(* Logix 5000 project; controller HP_SSC01 vendor 1 type 14 code 67 rev 17.7; software revision 17.01; part 6 of 15 *)
(* tags used below, declared in another part *)
   A_C2_0218 : ALIAS FOR S_C2_FaultSafety.18;
   A_C2_0219 : ALIAS FOR S_C2_FaultSafety.19;
   A_C2_0220 : ALIAS FOR S_C2_FaultSafety.20;
   A_C2_0221 : ALIAS FOR S_C2_FaultSafety.21;
   A_C2_0222 : ALIAS FOR S_C2_FaultSafety.22;
   A_C2_0223 : ALIAS FOR S_C2_FaultSafety.23;
   A_C2_0311 : ALIAS FOR C2_FaultStandard.11;
   A_C2_0312 : ALIAS FOR C2_FaultStandard.12;
   A_C2_0313 : ALIAS FOR C2_FaultStandard.13;
   A_C2_0314 : ALIAS FOR C2_FaultStandard.14;
   A_C2_0315 : ALIAS FOR C2_FaultStandard.15;
   C2 : AXIS_SERVO_DRIVE;
   C2_EncoderDegree : REAL;
   C2_EncoderPositionAtHome : DINT;
   C2_ExcecutePBHoldTimer : TIMER;
   C2_FaultHomeSwitchNotFound : BOOL;
   C2_Homed : BOOL;
   C2_HomeDelay : TIMER[8];
   C2_HomeFindSwitchMAM01 : MOTION_INSTRUCTION;
   C2_HomeFindSwitchMAM02 : MOTION_INSTRUCTION;
   C2_HomeFindSwitchMAS01 : MOTION_INSTRUCTION;
   C2_HomeGetCloseToSwitchMAM01 : MOTION_INSTRUCTION;
   C2_HomeGoToOnPathMAM01 : MOTION_INSTRUCTION;
   C2_HomeMessageNumber : DINT;
   C2_HomeSensorTestMAM02 : MOTION_INSTRUCTION;
   C2_HomeSequence : DINT;
   C2_HomeSequenceAlarms : DINT;
   C2_HomeSequenceAlarmTimer : TIMER[32];
   C2_HomeSequenceInProcess : BOOL;
   C2_HomeSequenceMAH : MOTION_INSTRUCTION;
   C2_HomeSwitchFaultK7KFailedOff : BOOL;
   C2_HomeSwitchFaultK7KFailedOn : BOOL;
   C2_HomeSwitchFaultSafeFailedOff : BOOL;
   C2_HomeSwitchFaultSafeFailedOn : BOOL;
   C2_HomeTest : REAL;
   C2_IndexEnable : BOOL;
   C2_IndexEnableTOF : TIMER;
   C2_IndexMAM01 : MOTION_INSTRUCTION;
   C2_IndexMAS01 : MOTION_INSTRUCTION;
   C2_IndexMessageNumber : DINT;
   C2_IndexPermissive : BOOL;
   C2_Jog_ONS : DINT;
   C2_JogDirection : DINT;
   C2_JogEnable : BOOL;
   C2_JogEnableTOF : TIMER;
   C2_JogForwardFastSelected : BOOL;
   C2_JogForwardSlowSelected : BOOL;
   C2_JogMAJ01 : MOTION_INSTRUCTION;
   C2_JogMAJ02 : MOTION_INSTRUCTION;
   C2_JogMAS01 : MOTION_INSTRUCTION;
   C2_JogMessageNumber : DINT;
   C2_JogPermissive : BOOL;
   C2_JogReverseFastSelected : BOOL;
   C2_JogReverseSlowSelected : BOOL;
   C2_MAJAcceleration : REAL;
   C2_MAJDeceleration : REAL;
   C2_MAJSpeed : REAL;
   C2_OIT_Current : DINT;
   C2_RemoteHomeCMD : BOOL;
   C2_ServoActionStatusOnDelay : TIMER;
   C2_SetEncoderHomePosition : BOOL;
   C2HomeSensorTestMAM01 : MOTION_INSTRUCTION;
   C2HomeSequenceONS : BOOL;
   C2HomeSequenceONS2 : BOOL;
   S_C2_EncoderPositionAtHomeSet : BOOL;
   S_C2_ExecutePB : BOOL;
   S_C2_FaultReset : BOOL;
   S_C2_HomeSafePE : ALIAS FOR C2_Safe:I.Pt04Data;
   S_C2_ModeLocal : BOOL;
   S_C2_ModeRemote : BOOL;
   S_C2_MSTOP_InputOK : BOOL;
   S_EncoderCtsFor360Deg : DINT;
(* Carousel2, continued *)

ROUTINE C230_Home   (* ladder *)
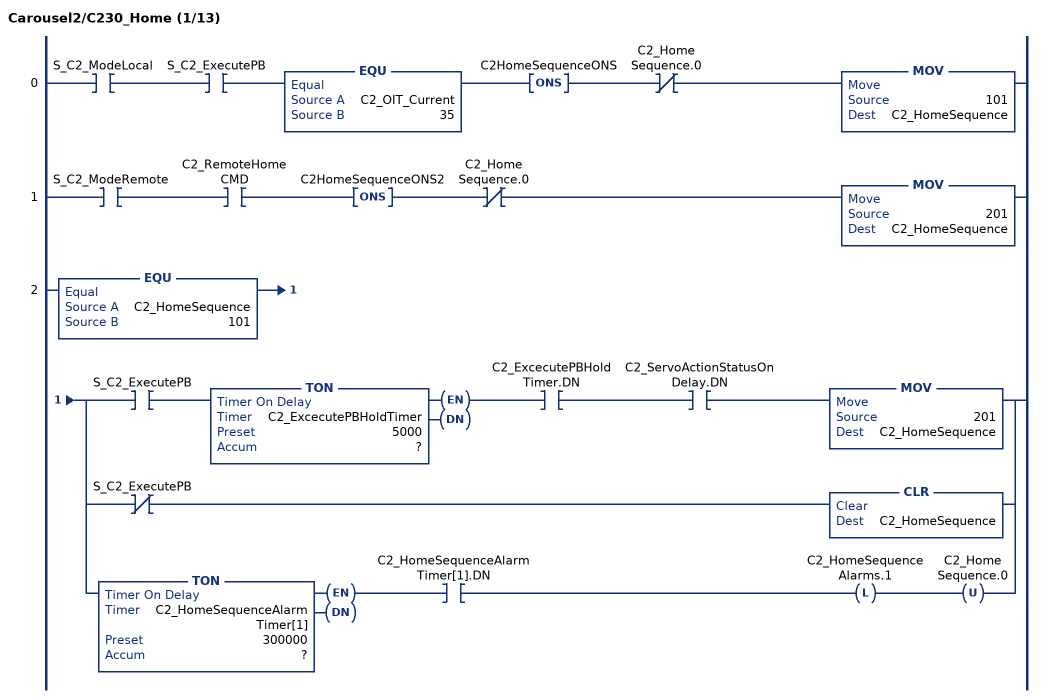
   0: XIC(S_C2_ModeLocal)XIC(S_C2_ExecutePB)EQU(C2_OIT_Current,35)ONS(C2HomeSequenceONS)XIO(C2_HomeSequence.0)MOV(101,C2_HomeSequence);
   1: XIC(S_C2_ModeRemote)XIC(C2_RemoteHomeCMD)ONS(C2HomeSequenceONS2)XIO(C2_HomeSequence.0)MOV(201,C2_HomeSequence);
   2: EQU(C2_HomeSequence,101)[XIC(S_C2_ExecutePB) TON(C2_ExcecutePBHoldTimer,?,?) XIC(C2_ExcecutePBHoldTimer.DN) XIC(C2_ServoActionStatusOnDelay.DN) MOV(201,C2_HomeSequence) ,XIO(S_C2_ExecutePB) CLR(C2_HomeSequence) ,TON(C2_HomeSequenceAlarmTimer[1],?,?) XIC(C2_HomeSequenceAlarmTimer[1].DN) OTL(C2_HomeSequenceAlarms.1) OTU(C2_HomeSequence.0) ];
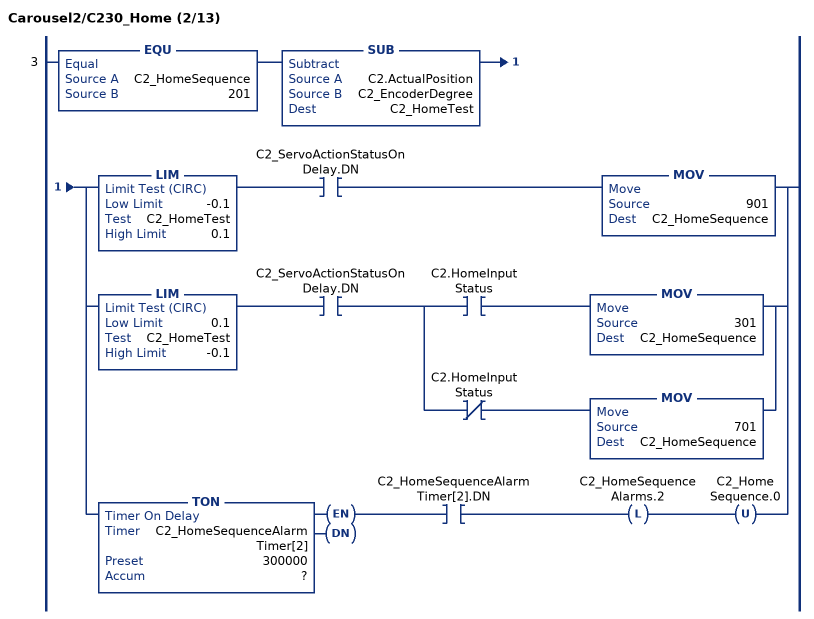
   3: EQU(C2_HomeSequence,201)SUB(C2.ActualPosition,C2_EncoderDegree,C2_HomeTest)[LIM(-0.1,C2_HomeTest,0.1) XIC(C2_ServoActionStatusOnDelay.DN) MOV(901,C2_HomeSequence) ,LIM(0.1,C2_HomeTest,-0.1) XIC(C2_ServoActionStatusOnDelay.DN) [XIC(C2.HomeInputStatus) MOV(301,C2_HomeSequence) ,XIO(C2.HomeInputStatus) MOV(701,C2_HomeSequence) ] ,TON(C2_HomeSequenceAlarmTimer[2],?,?) XIC(C2_HomeSequenceAlarmTimer[2].DN) OTL(C2_HomeSequenceAlarms.2) OTU(C2_HomeSequence.0) ];
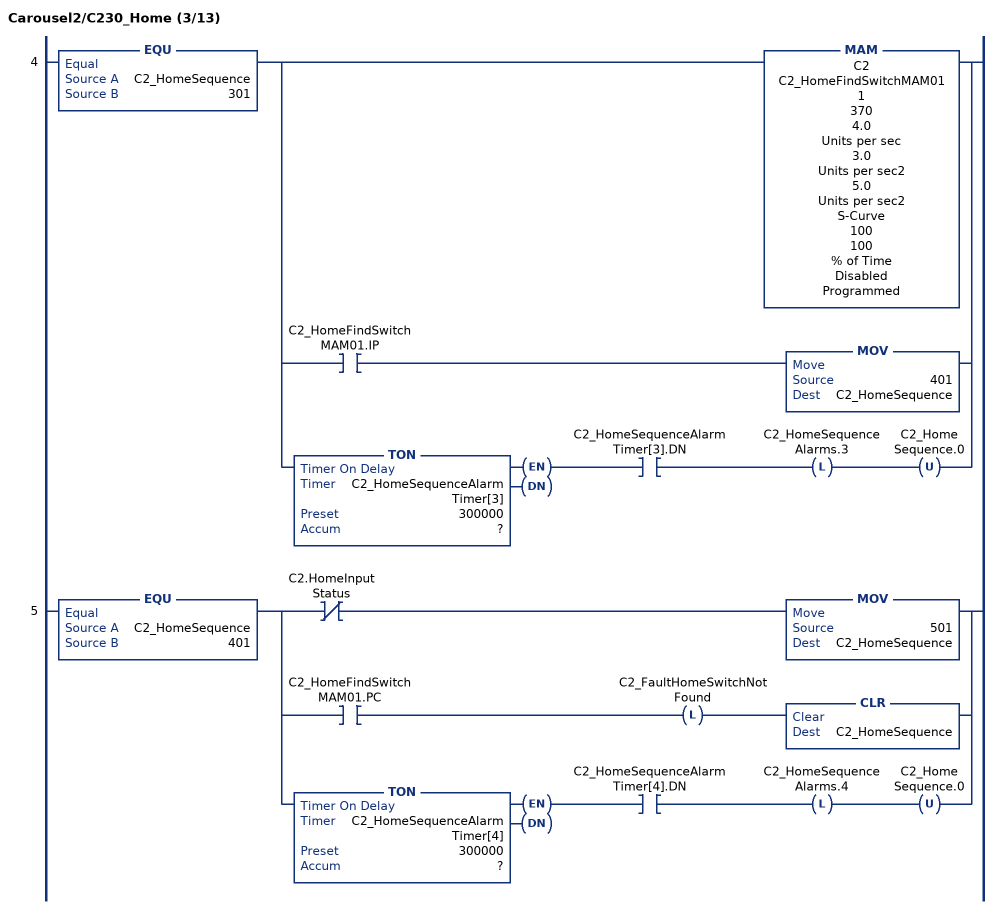
   4: EQU(C2_HomeSequence,301)[MAM(C2,C2_HomeFindSwitchMAM01,1,370,4.0,Units per sec,3.0,Units per sec2,5.0,Units per sec2,S-Curve,100,100,% of Time,Disabled,Programmed) ,XIC(C2_HomeFindSwitchMAM01.IP) MOV(401,C2_HomeSequence) ,TON(C2_HomeSequenceAlarmTimer[3],?,?) XIC(C2_HomeSequenceAlarmTimer[3].DN) OTL(C2_HomeSequenceAlarms.3) OTU(C2_HomeSequence.0) ];
   5: EQU(C2_HomeSequence,401)[XIO(C2.HomeInputStatus) MOV(501,C2_HomeSequence) ,XIC(C2_HomeFindSwitchMAM01.PC) OTL(C2_FaultHomeSwitchNotFound) CLR(C2_HomeSequence) ,TON(C2_HomeSequenceAlarmTimer[4],?,?) XIC(C2_HomeSequenceAlarmTimer[4].DN) OTL(C2_HomeSequenceAlarms.4) OTU(C2_HomeSequence.0) ];
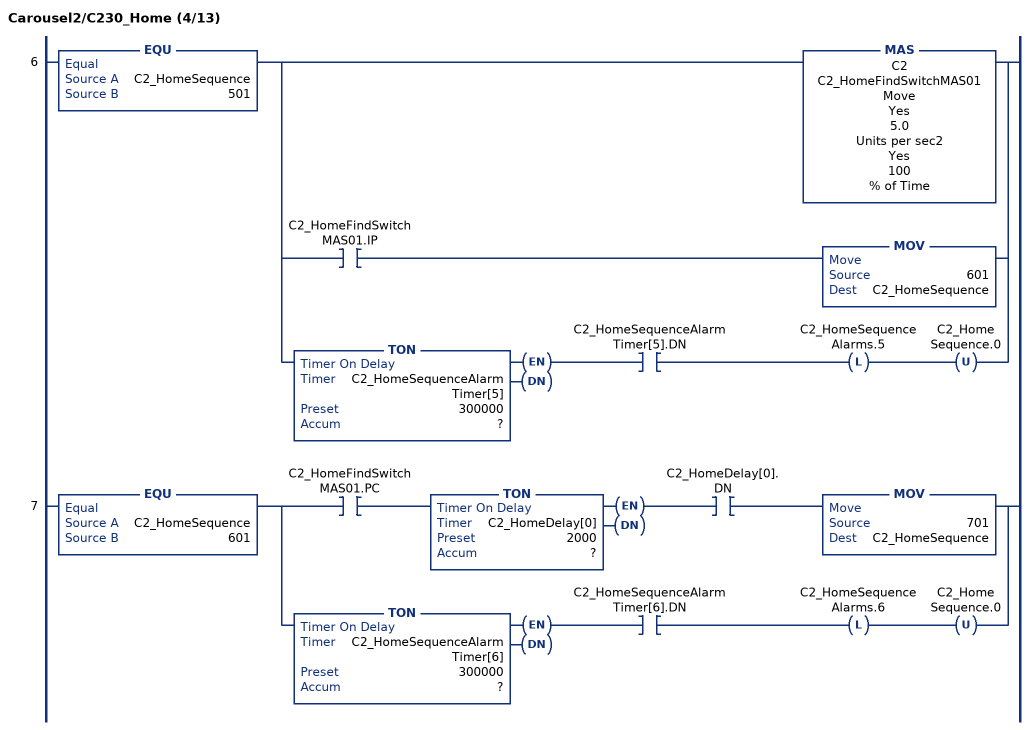
   6: EQU(C2_HomeSequence,501)[MAS(C2,C2_HomeFindSwitchMAS01,Move,Yes,5.0,Units per sec2,Yes,100,% of Time) ,XIC(C2_HomeFindSwitchMAS01.IP) MOV(601,C2_HomeSequence) ,TON(C2_HomeSequenceAlarmTimer[5],?,?) XIC(C2_HomeSequenceAlarmTimer[5].DN) OTL(C2_HomeSequenceAlarms.5) OTU(C2_HomeSequence.0) ];
   7: EQU(C2_HomeSequence,601)[XIC(C2_HomeFindSwitchMAS01.PC) TON(C2_HomeDelay[0],?,?) XIC(C2_HomeDelay[0].DN) MOV(701,C2_HomeSequence) ,TON(C2_HomeSequenceAlarmTimer[6],?,?) XIC(C2_HomeSequenceAlarmTimer[6].DN) OTL(C2_HomeSequenceAlarms.6) OTU(C2_HomeSequence.0) ];
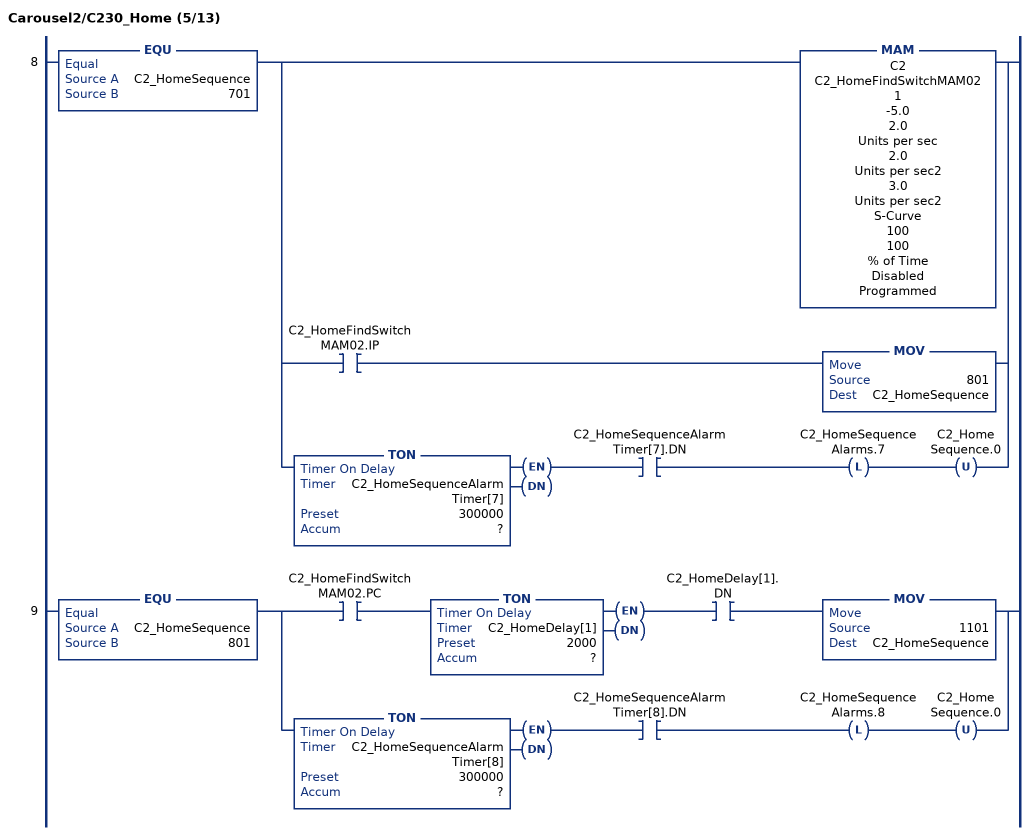
   8: EQU(C2_HomeSequence,701)[MAM(C2,C2_HomeFindSwitchMAM02,1,-5.0,2.0,Units per sec,2.0,Units per sec2,3.0,Units per sec2,S-Curve,100,100,% of Time,Disabled,Programmed) ,XIC(C2_HomeFindSwitchMAM02.IP) MOV(801,C2_HomeSequence) ,TON(C2_HomeSequenceAlarmTimer[7],?,?) XIC(C2_HomeSequenceAlarmTimer[7].DN) OTL(C2_HomeSequenceAlarms.7) OTU(C2_HomeSequence.0) ];
   9: EQU(C2_HomeSequence,801)[XIC(C2_HomeFindSwitchMAM02.PC) TON(C2_HomeDelay[1],?,?) XIC(C2_HomeDelay[1].DN) MOV(1101,C2_HomeSequence) ,TON(C2_HomeSequenceAlarmTimer[8],?,?) XIC(C2_HomeSequenceAlarmTimer[8].DN) OTL(C2_HomeSequenceAlarms.8) OTU(C2_HomeSequence.0) ];
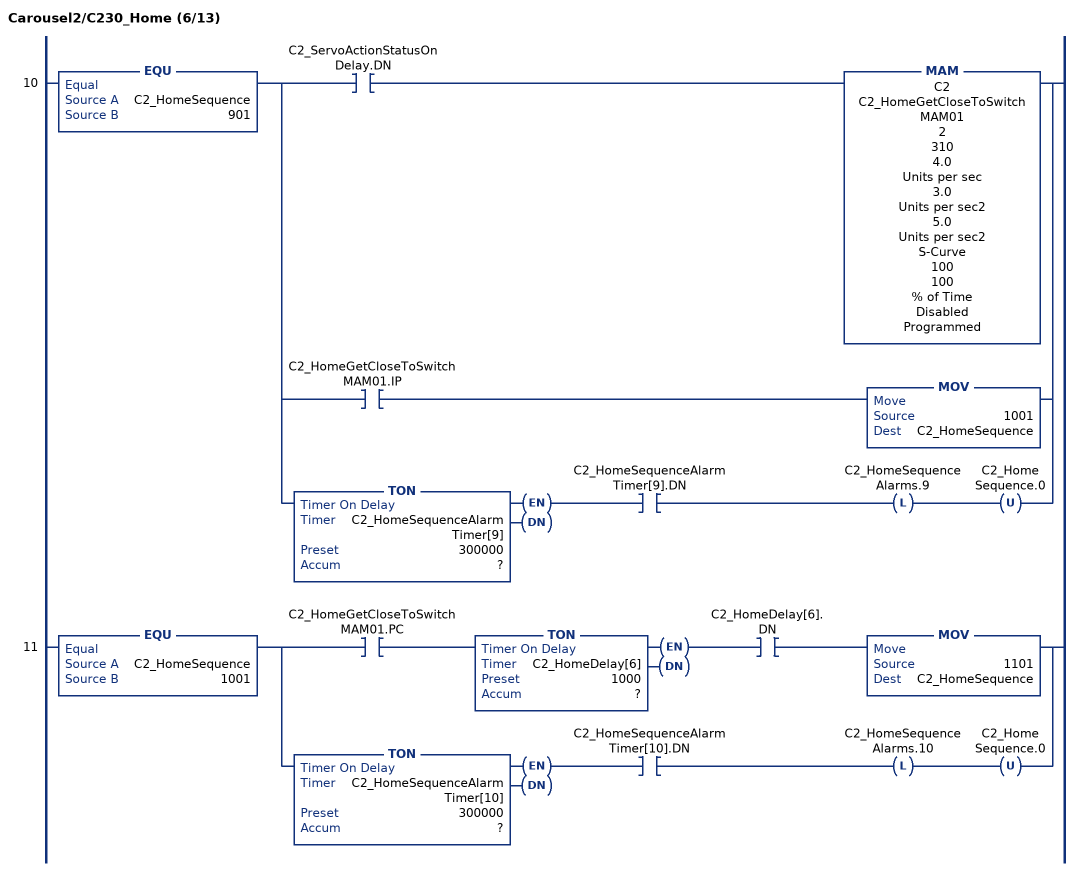
   10: EQU(C2_HomeSequence,901)[XIC(C2_ServoActionStatusOnDelay.DN) MAM(C2,C2_HomeGetCloseToSwitchMAM01,2,310,4.0,Units per sec,3.0,Units per sec2,5.0,Units per sec2,S-Curve,100,100,% of Time,Disabled,Programmed) ,XIC(C2_HomeGetCloseToSwitchMAM01.IP) MOV(1001,C2_HomeSequence) ,TON(C2_HomeSequenceAlarmTimer[9],?,?) XIC(C2_HomeSequenceAlarmTimer[9].DN) OTL(C2_HomeSequenceAlarms.9) OTU(C2_HomeSequence.0) ];
   11: EQU(C2_HomeSequence,1001)[XIC(C2_HomeGetCloseToSwitchMAM01.PC) TON(C2_HomeDelay[6],?,?) XIC(C2_HomeDelay[6].DN) MOV(1101,C2_HomeSequence) ,TON(C2_HomeSequenceAlarmTimer[10],?,?) XIC(C2_HomeSequenceAlarmTimer[10].DN) OTL(C2_HomeSequenceAlarms.10) OTU(C2_HomeSequence.0) ];
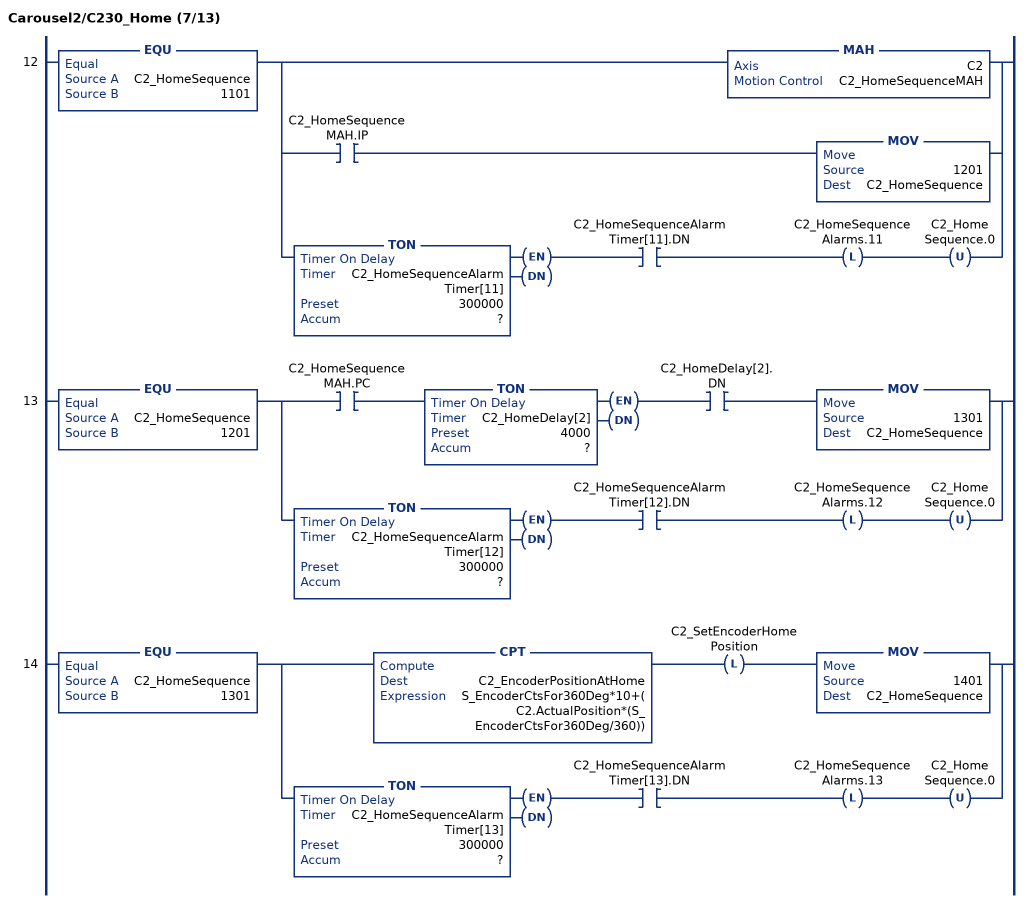
   12: EQU(C2_HomeSequence,1101)[MAH(C2,C2_HomeSequenceMAH) ,XIC(C2_HomeSequenceMAH.IP) MOV(1201,C2_HomeSequence) ,TON(C2_HomeSequenceAlarmTimer[11],?,?) XIC(C2_HomeSequenceAlarmTimer[11].DN) OTL(C2_HomeSequenceAlarms.11) OTU(C2_HomeSequence.0) ];
   13: EQU(C2_HomeSequence,1201)[XIC(C2_HomeSequenceMAH.PC) TON(C2_HomeDelay[2],?,?) XIC(C2_HomeDelay[2].DN) MOV(1301,C2_HomeSequence) ,TON(C2_HomeSequenceAlarmTimer[12],?,?) XIC(C2_HomeSequenceAlarmTimer[12].DN) OTL(C2_HomeSequenceAlarms.12) OTU(C2_HomeSequence.0) ];
   14: EQU(C2_HomeSequence,1301)[CPT(C2_EncoderPositionAtHome,S_EncoderCtsFor360Deg*10+(C2.ActualPosition*(S_EncoderCtsFor360Deg/360))) OTL(C2_SetEncoderHomePosition) MOV(1401,C2_HomeSequence) ,TON(C2_HomeSequenceAlarmTimer[13],?,?) XIC(C2_HomeSequenceAlarmTimer[13].DN) OTL(C2_HomeSequenceAlarms.13) OTU(C2_HomeSequence.0) ];
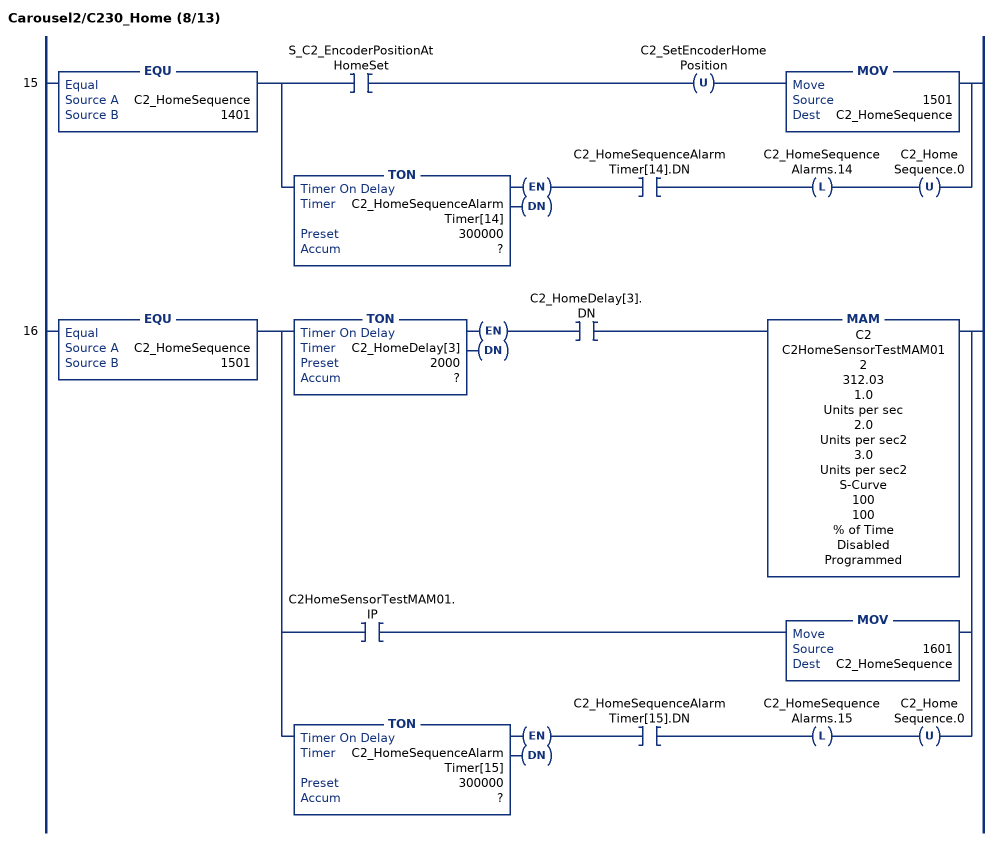
   15: EQU(C2_HomeSequence,1401)[XIC(S_C2_EncoderPositionAtHomeSet) OTU(C2_SetEncoderHomePosition) MOV(1501,C2_HomeSequence) ,TON(C2_HomeSequenceAlarmTimer[14],?,?) XIC(C2_HomeSequenceAlarmTimer[14].DN) OTL(C2_HomeSequenceAlarms.14) OTU(C2_HomeSequence.0) ];
   16: EQU(C2_HomeSequence,1501)[TON(C2_HomeDelay[3],?,?) XIC(C2_HomeDelay[3].DN) MAM(C2,C2HomeSensorTestMAM01,2,312.03,1.0,Units per sec,2.0,Units per sec2,3.0,Units per sec2,S-Curve,100,100,% of Time,Disabled,Programmed) ,XIC(C2HomeSensorTestMAM01.IP) MOV(1601,C2_HomeSequence) ,TON(C2_HomeSequenceAlarmTimer[15],?,?) XIC(C2_HomeSequenceAlarmTimer[15].DN) OTL(C2_HomeSequenceAlarms.15) OTU(C2_HomeSequence.0) ];
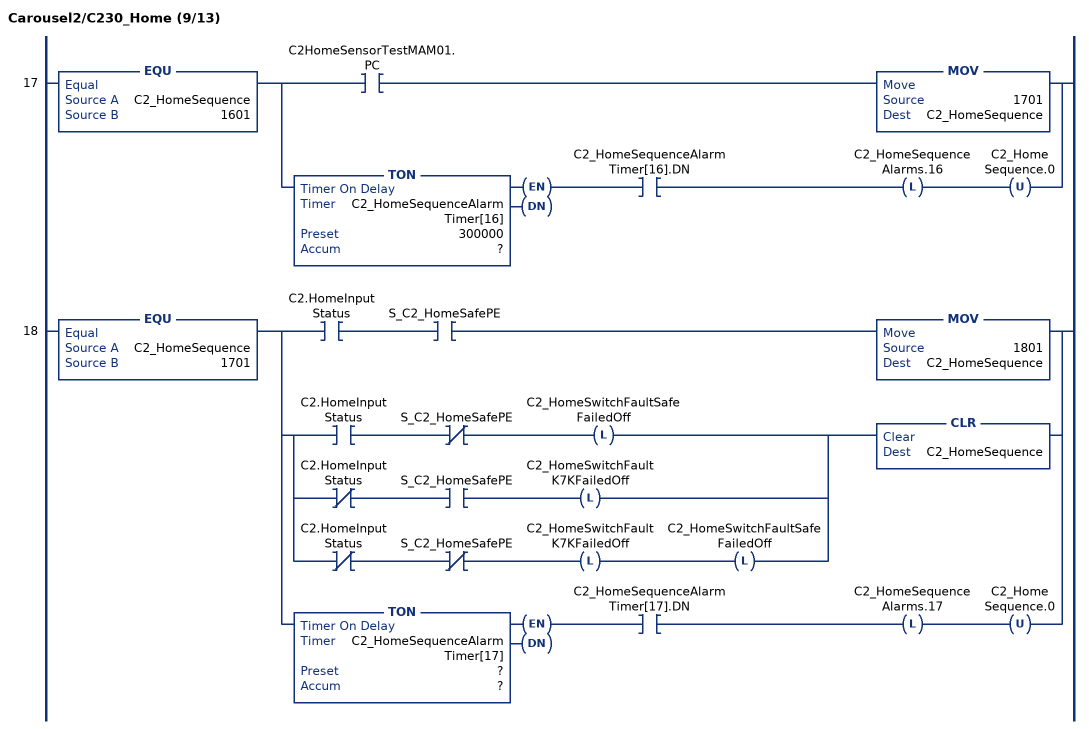
   17: EQU(C2_HomeSequence,1601)[XIC(C2HomeSensorTestMAM01.PC) MOV(1701,C2_HomeSequence) ,TON(C2_HomeSequenceAlarmTimer[16],?,?) XIC(C2_HomeSequenceAlarmTimer[16].DN) OTL(C2_HomeSequenceAlarms.16) OTU(C2_HomeSequence.0) ];
   18: EQU(C2_HomeSequence,1701)[XIC(C2.HomeInputStatus) XIC(S_C2_HomeSafePE) MOV(1801,C2_HomeSequence) ,[XIC(C2.HomeInputStatus) XIO(S_C2_HomeSafePE) OTL(C2_HomeSwitchFaultSafeFailedOff) ,XIO(C2.HomeInputStatus) XIC(S_C2_HomeSafePE) OTL(C2_HomeSwitchFaultK7KFailedOff) ,XIO(C2.HomeInputStatus) XIO(S_C2_HomeSafePE) OTL(C2_HomeSwitchFaultK7KFailedOff) OTL(C2_HomeSwitchFaultSafeFailedOff) ] CLR(C2_HomeSequence) ,TON(C2_HomeSequenceAlarmTimer[17],?,?) XIC(C2_HomeSequenceAlarmTimer[17].DN) OTL(C2_HomeSequenceAlarms.17) OTU(C2_HomeSequence.0) ];
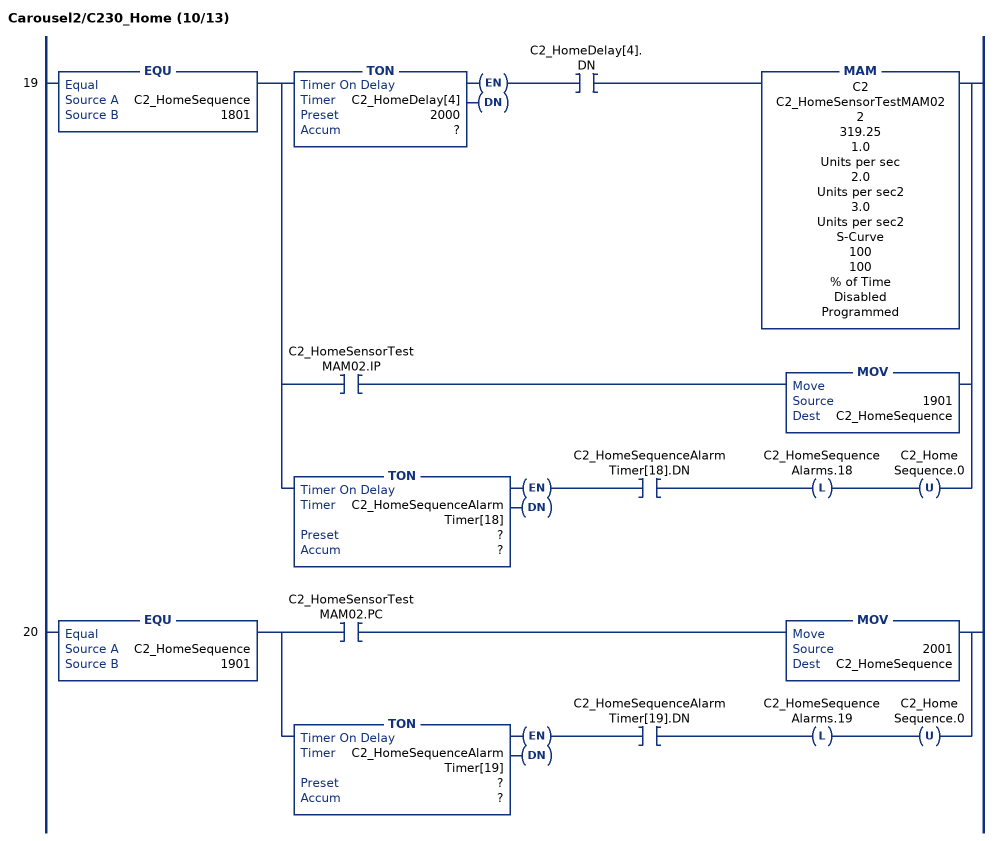
   19: EQU(C2_HomeSequence,1801)[TON(C2_HomeDelay[4],?,?) XIC(C2_HomeDelay[4].DN) MAM(C2,C2_HomeSensorTestMAM02,2,319.25,1.0,Units per sec,2.0,Units per sec2,3.0,Units per sec2,S-Curve,100,100,% of Time,Disabled,Programmed) ,XIC(C2_HomeSensorTestMAM02.IP) MOV(1901,C2_HomeSequence) ,TON(C2_HomeSequenceAlarmTimer[18],?,?) XIC(C2_HomeSequenceAlarmTimer[18].DN) OTL(C2_HomeSequenceAlarms.18) OTU(C2_HomeSequence.0) ];
   20: EQU(C2_HomeSequence,1901)[XIC(C2_HomeSensorTestMAM02.PC) MOV(2001,C2_HomeSequence) ,TON(C2_HomeSequenceAlarmTimer[19],?,?) XIC(C2_HomeSequenceAlarmTimer[19].DN) OTL(C2_HomeSequenceAlarms.19) OTU(C2_HomeSequence.0) ];
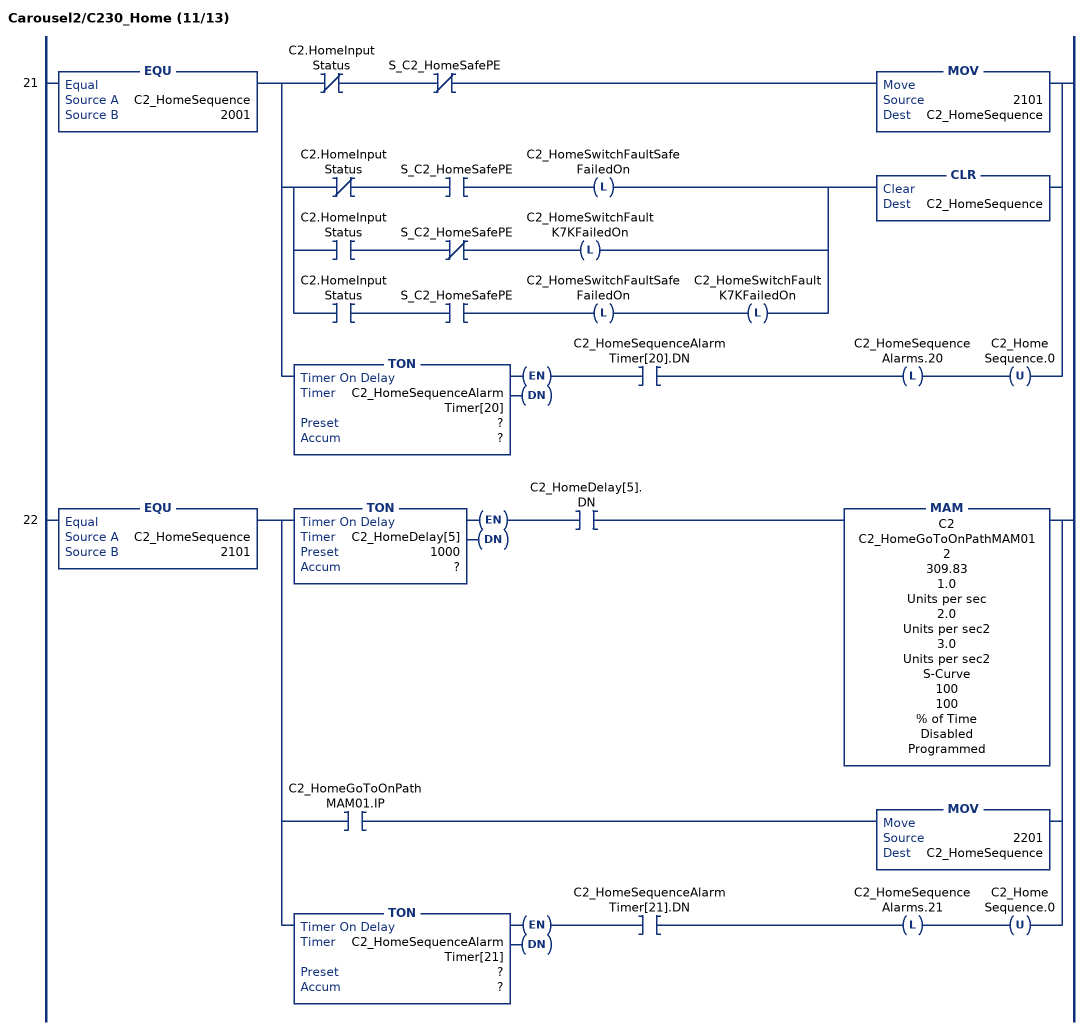
   21: EQU(C2_HomeSequence,2001)[XIO(C2.HomeInputStatus) XIO(S_C2_HomeSafePE) MOV(2101,C2_HomeSequence) ,[XIO(C2.HomeInputStatus) XIC(S_C2_HomeSafePE) OTL(C2_HomeSwitchFaultSafeFailedOn) ,XIC(C2.HomeInputStatus) XIO(S_C2_HomeSafePE) OTL(C2_HomeSwitchFaultK7KFailedOn) ,XIC(C2.HomeInputStatus) XIC(S_C2_HomeSafePE) OTL(C2_HomeSwitchFaultSafeFailedOn) OTL(C2_HomeSwitchFaultK7KFailedOn) ] CLR(C2_HomeSequence) ,TON(C2_HomeSequenceAlarmTimer[20],?,?) XIC(C2_HomeSequenceAlarmTimer[20].DN) OTL(C2_HomeSequenceAlarms.20) OTU(C2_HomeSequence.0) ];
   22: EQU(C2_HomeSequence,2101)[TON(C2_HomeDelay[5],?,?) XIC(C2_HomeDelay[5].DN) MAM(C2,C2_HomeGoToOnPathMAM01,2,309.83,1.0,Units per sec,2.0,Units per sec2,3.0,Units per sec2,S-Curve,100,100,% of Time,Disabled,Programmed) ,XIC(C2_HomeGoToOnPathMAM01.IP) MOV(2201,C2_HomeSequence) ,TON(C2_HomeSequenceAlarmTimer[21],?,?) XIC(C2_HomeSequenceAlarmTimer[21].DN) OTL(C2_HomeSequenceAlarms.21) OTU(C2_HomeSequence.0) ];
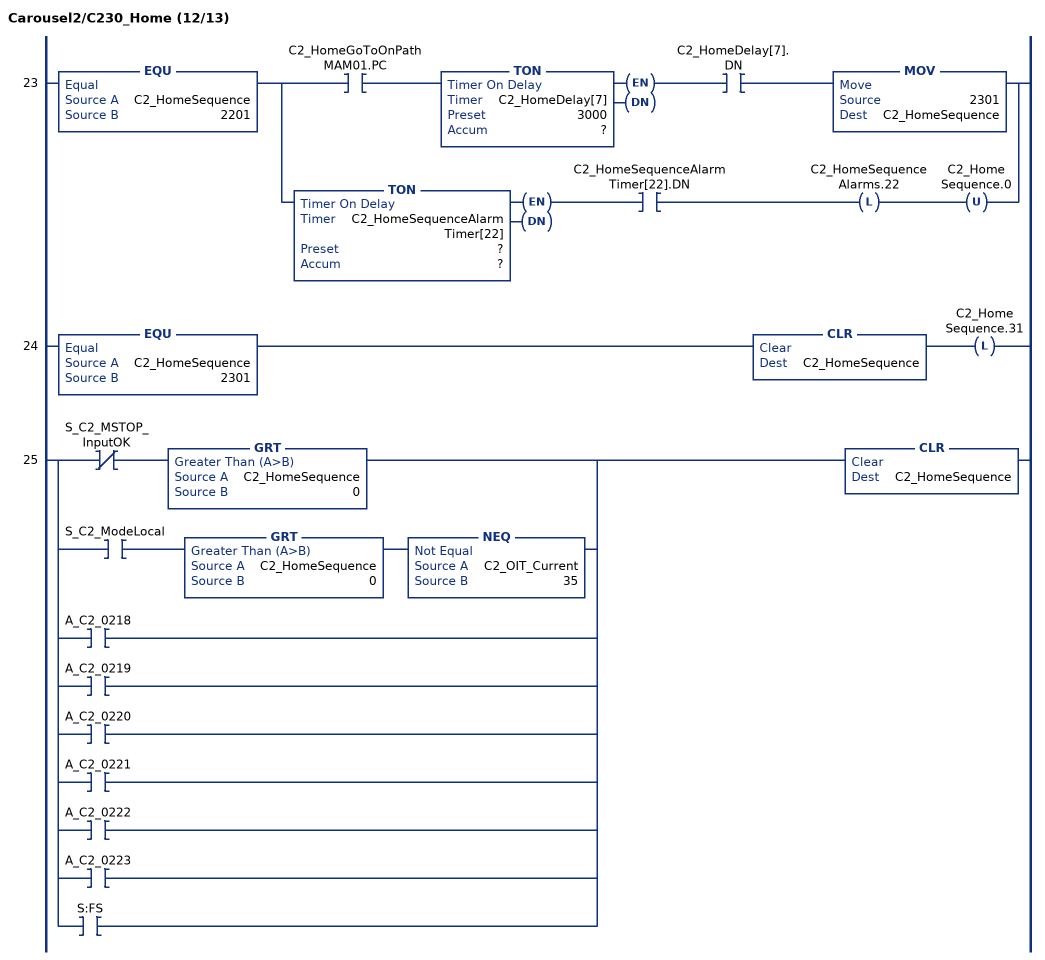
   23: EQU(C2_HomeSequence,2201)[XIC(C2_HomeGoToOnPathMAM01.PC) TON(C2_HomeDelay[7],?,?) XIC(C2_HomeDelay[7].DN) MOV(2301,C2_HomeSequence) ,TON(C2_HomeSequenceAlarmTimer[22],?,?) XIC(C2_HomeSequenceAlarmTimer[22].DN) OTL(C2_HomeSequenceAlarms.22) OTU(C2_HomeSequence.0) ];
   24: EQU(C2_HomeSequence,2301)CLR(C2_HomeSequence)OTL(C2_HomeSequence.31);
   25: [XIO(S_C2_MSTOP_InputOK) GRT(C2_HomeSequence,0) ,XIC(S_C2_ModeLocal) GRT(C2_HomeSequence,0) NEQ(C2_OIT_Current,35) ,XIC(A_C2_0218) ,XIC(A_C2_0219) ,XIC(A_C2_0220) ,XIC(A_C2_0221) ,XIC(A_C2_0222) ,XIC(A_C2_0223) ,XIC(S:FS) ]CLR(C2_HomeSequence);
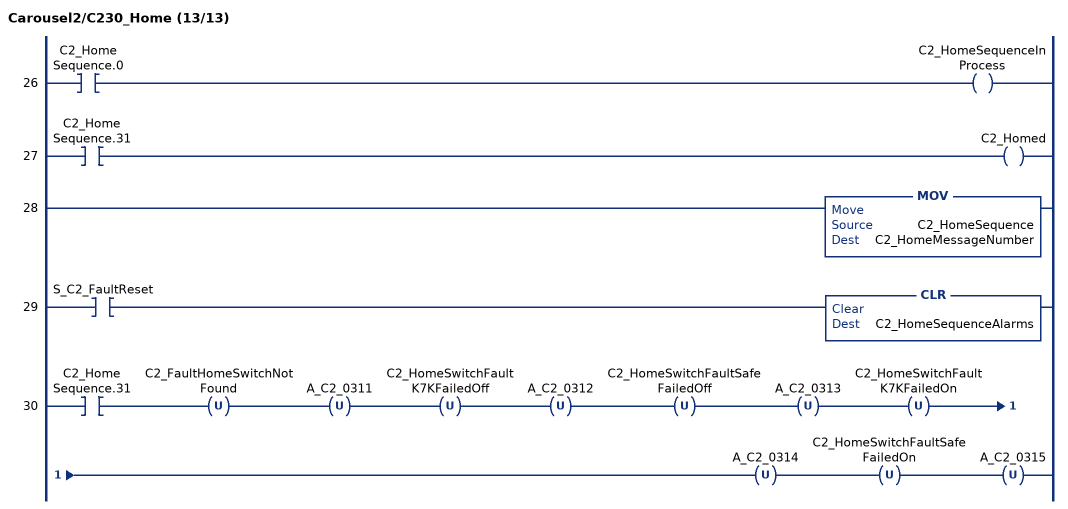
   26: XIC(C2_HomeSequence.0)OTE(C2_HomeSequenceInProcess);
   27: XIC(C2_HomeSequence.31)OTE(C2_Homed);
   28: MOV(C2_HomeSequence,C2_HomeMessageNumber);
   29: XIC(S_C2_FaultReset)CLR(C2_HomeSequenceAlarms);
   30: XIC(C2_HomeSequence.31)OTU(C2_FaultHomeSwitchNotFound)OTU(A_C2_0311)OTU(C2_HomeSwitchFaultK7KFailedOff)OTU(A_C2_0312)OTU(C2_HomeSwitchFaultSafeFailedOff)OTU(A_C2_0313)OTU(C2_HomeSwitchFaultK7KFailedOn)OTU(A_C2_0314)OTU(C2_HomeSwitchFaultSafeFailedOn)OTU(A_C2_0315);
END_ROUTINE

ROUTINE C235_Index   (* ladder *)
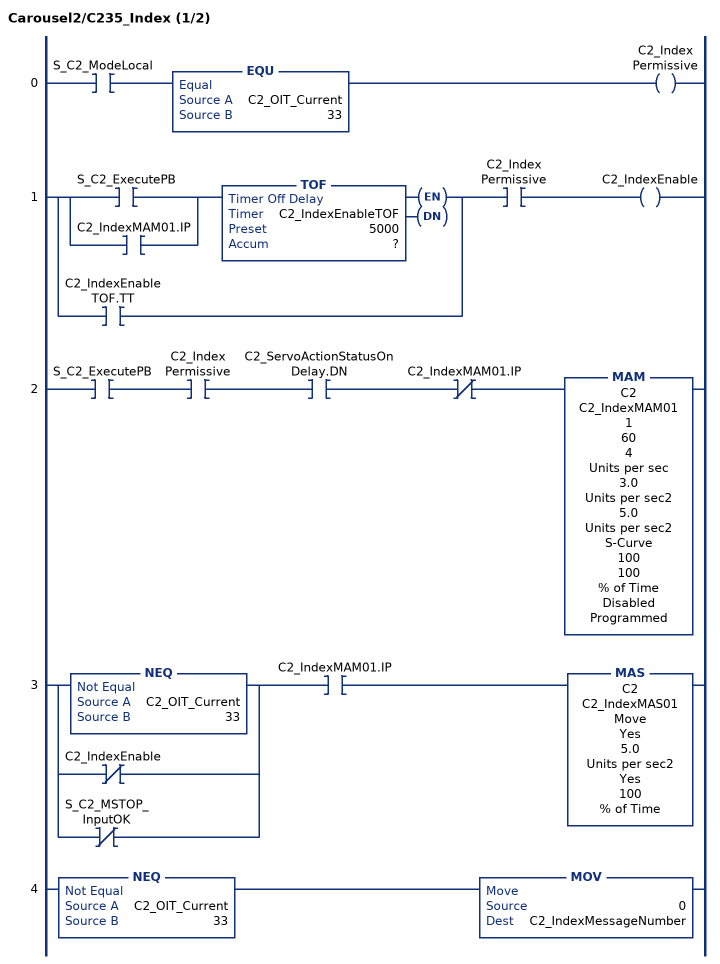
   0: XIC(S_C2_ModeLocal)EQU(C2_OIT_Current,33)OTE(C2_IndexPermissive);
   1: [[XIC(S_C2_ExecutePB) ,XIC(C2_IndexMAM01.IP) ] TOF(C2_IndexEnableTOF,?,?) ,XIC(C2_IndexEnableTOF.TT) ]XIC(C2_IndexPermissive)OTE(C2_IndexEnable);
   2: XIC(S_C2_ExecutePB)XIC(C2_IndexPermissive)XIC(C2_ServoActionStatusOnDelay.DN)XIO(C2_IndexMAM01.IP)MAM(C2,C2_IndexMAM01,1,60,4,Units per sec,3.0,Units per sec2,5.0,Units per sec2,S-Curve,100,100,% of Time,Disabled,Programmed);
   3: [NEQ(C2_OIT_Current,33) ,XIO(C2_IndexEnable) ,XIO(S_C2_MSTOP_InputOK) ]XIC(C2_IndexMAM01.IP)MAS(C2,C2_IndexMAS01,Move,Yes,5.0,Units per sec2,Yes,100,% of Time);
   4: NEQ(C2_OIT_Current,33)MOV(0,C2_IndexMessageNumber);
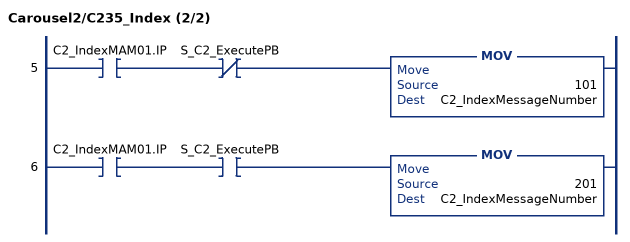
   5: XIC(C2_IndexMAM01.IP)XIO(S_C2_ExecutePB)MOV(101,C2_IndexMessageNumber);
   6: XIC(C2_IndexMAM01.IP)XIC(S_C2_ExecutePB)MOV(201,C2_IndexMessageNumber);
END_ROUTINE

ROUTINE C240_Jog   (* ladder *)
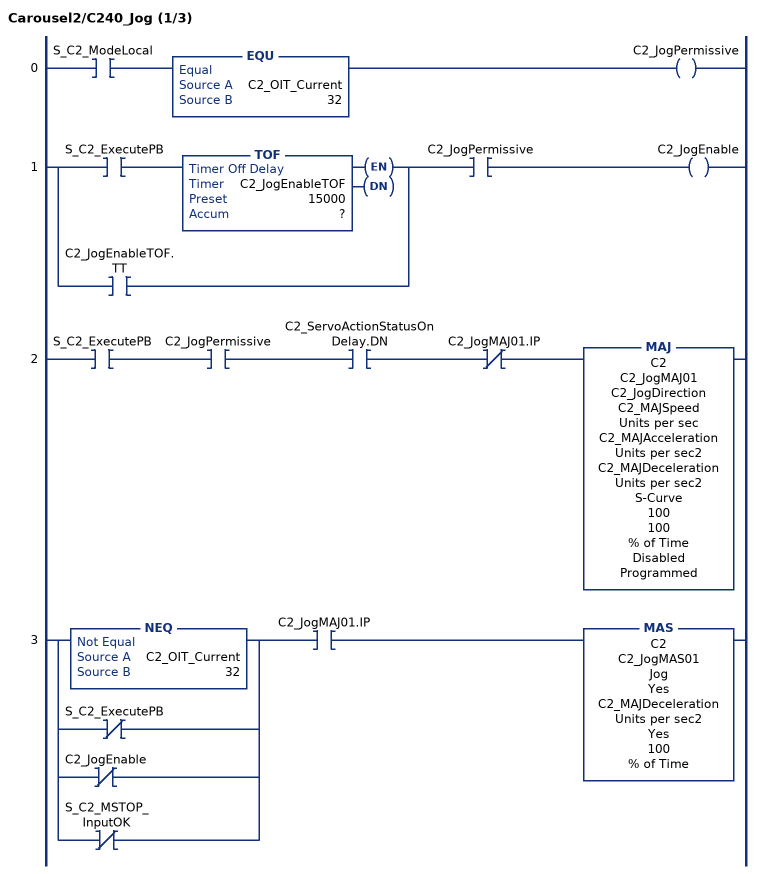
   0: XIC(S_C2_ModeLocal)EQU(C2_OIT_Current,32)OTE(C2_JogPermissive);
   1: [XIC(S_C2_ExecutePB) TOF(C2_JogEnableTOF,?,?) ,XIC(C2_JogEnableTOF.TT) ]XIC(C2_JogPermissive)OTE(C2_JogEnable);
   2: XIC(S_C2_ExecutePB)XIC(C2_JogPermissive)XIC(C2_ServoActionStatusOnDelay.DN)XIO(C2_JogMAJ01.IP)MAJ(C2,C2_JogMAJ01,C2_JogDirection,C2_MAJSpeed,Units per sec,C2_MAJAcceleration,Units per sec2,C2_MAJDeceleration,Units per sec2,S-Curve,100,100,% of Time,Disabled,Programmed);
   3: [NEQ(C2_OIT_Current,32) ,XIO(S_C2_ExecutePB) ,XIO(C2_JogEnable) ,XIO(S_C2_MSTOP_InputOK) ]XIC(C2_JogMAJ01.IP)MAS(C2,C2_JogMAS01,Jog,Yes,C2_MAJDeceleration,Units per sec2,Yes,100,% of Time);
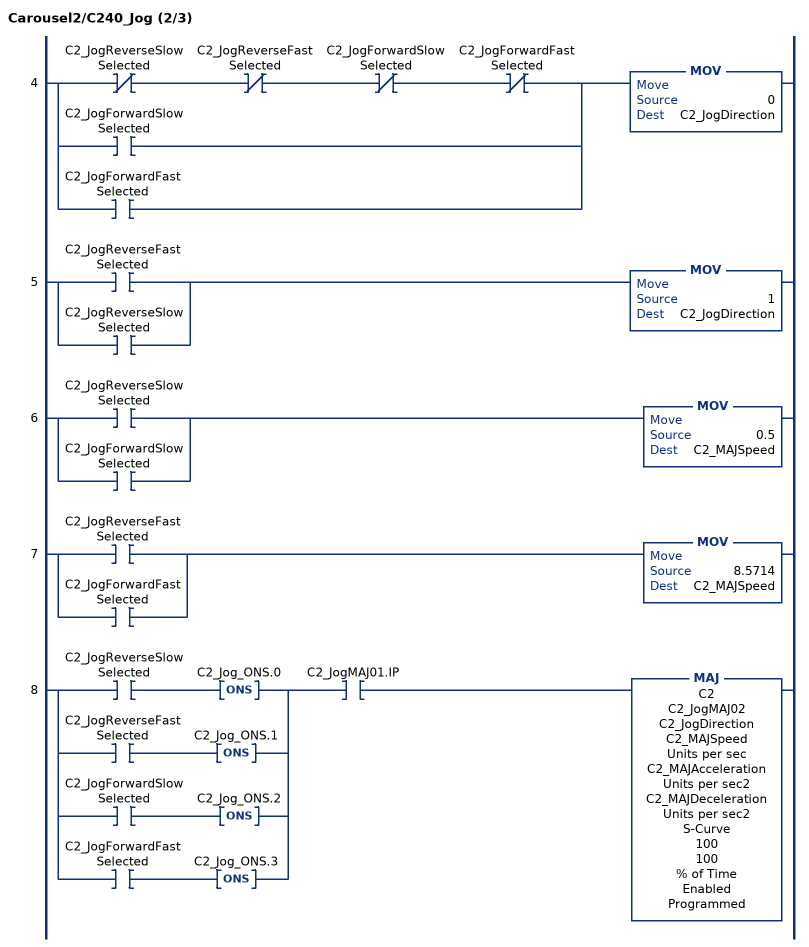
   4: [XIO(C2_JogReverseSlowSelected) XIO(C2_JogReverseFastSelected) XIO(C2_JogForwardSlowSelected) XIO(C2_JogForwardFastSelected) ,XIC(C2_JogForwardSlowSelected) ,XIC(C2_JogForwardFastSelected) ]MOV(0,C2_JogDirection);
   5: [XIC(C2_JogReverseFastSelected) ,XIC(C2_JogReverseSlowSelected) ]MOV(1,C2_JogDirection);
   6: [XIC(C2_JogReverseSlowSelected) ,XIC(C2_JogForwardSlowSelected) ]MOV(0.5,C2_MAJSpeed);
   7: [XIC(C2_JogReverseFastSelected) ,XIC(C2_JogForwardFastSelected) ]MOV(8.5714,C2_MAJSpeed);
   8: [XIC(C2_JogReverseSlowSelected) ONS(C2_Jog_ONS.0) ,XIC(C2_JogReverseFastSelected) ONS(C2_Jog_ONS.1) ,XIC(C2_JogForwardSlowSelected) ONS(C2_Jog_ONS.2) ,XIC(C2_JogForwardFastSelected) ONS(C2_Jog_ONS.3) ]XIC(C2_JogMAJ01.IP)MAJ(C2,C2_JogMAJ02,C2_JogDirection,C2_MAJSpeed,Units per sec,C2_MAJAcceleration,Units per sec2,C2_MAJDeceleration,Units per sec2,S-Curve,100,100,% of Time,Enabled,Programmed);
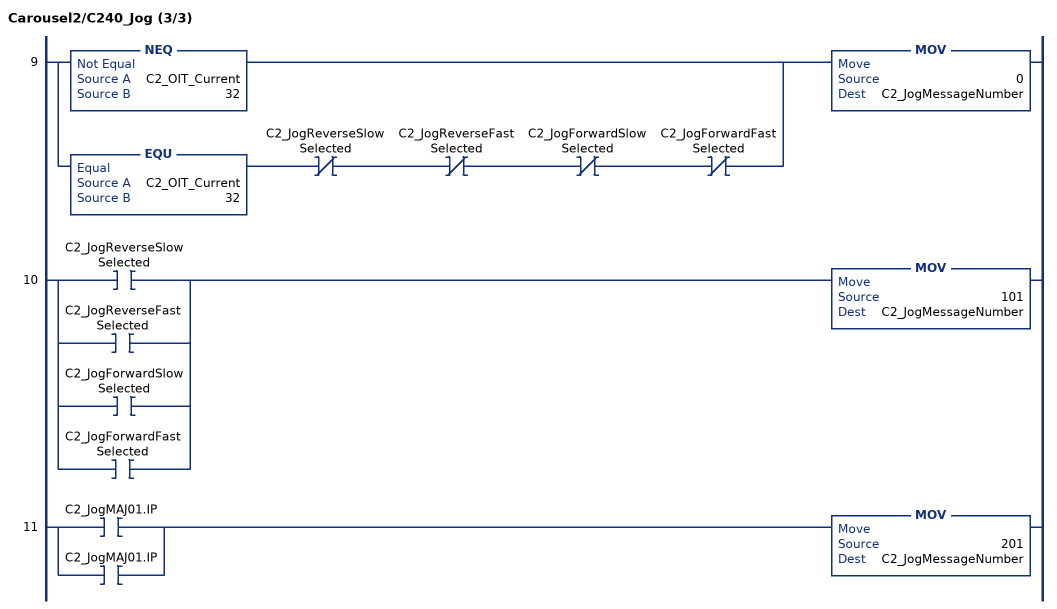
   9: [NEQ(C2_OIT_Current,32) ,EQU(C2_OIT_Current,32) XIO(C2_JogReverseSlowSelected) XIO(C2_JogReverseFastSelected) XIO(C2_JogForwardSlowSelected) XIO(C2_JogForwardFastSelected) ]MOV(0,C2_JogMessageNumber);
   10: [XIC(C2_JogReverseSlowSelected) ,XIC(C2_JogReverseFastSelected) ,XIC(C2_JogForwardSlowSelected) ,XIC(C2_JogForwardFastSelected) ]MOV(101,C2_JogMessageNumber);
   11: [XIC(C2_JogMAJ01.IP) ,XIC(C2_JogMAJ01.IP) ]MOV(201,C2_JogMessageNumber);
END_ROUTINE
